FUNCTION_BLOCK FB_FMS205_F2SeqPrep_SFC EXTENDS FB_ControllerBase_SFC
// Girar 8 veces el plato para determinar qué tipo de tapa hay en cada sector del plato

VAR_IN_OUT
	Medid			: FB_MedidorTapa;
	Induc		 	: FB_CaptadorInductivo;
	Fotoe			: FB_DetectorFotoelectrico;
	Plato			: FB_PlatoDivisor;
END_VAR

VAR
	Giros 			: INT := 0;
END_VAR

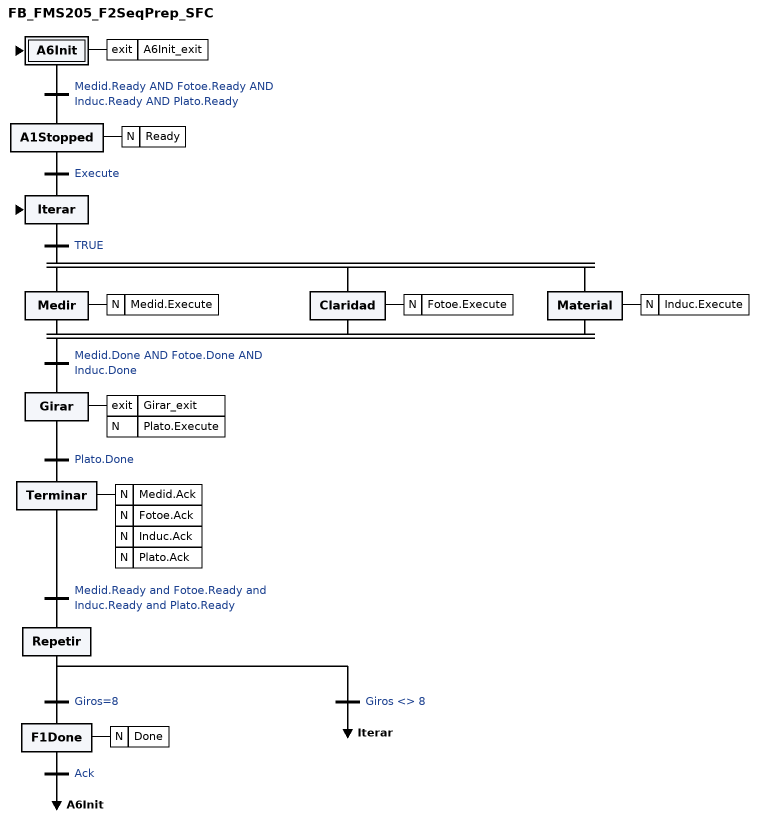
INITIAL_STEP A6Init:
    A6Init_exit(P0);  // exit action
END_STEP
TRANSITION FROM A6Init TO A1Stopped
    := Medid.Ready AND Fotoe.Ready AND Induc.Ready AND Plato.Ready;
END_TRANSITION
STEP A1Stopped:
    Ready(N);
END_STEP
TRANSITION FROM A1Stopped TO Iterar
    := Execute;
END_TRANSITION
STEP Iterar:
END_STEP
TRANSITION FROM Iterar TO (Medir, Claridad, Material)
    := TRUE;
END_TRANSITION
STEP Medir:
    Medid.Execute(N);
END_STEP
STEP Claridad:
    Fotoe.Execute(N);
END_STEP
STEP Material:
    Induc.Execute(N);
END_STEP
TRANSITION FROM (Medir, Claridad, Material) TO Girar
    := Medid.Done AND Fotoe.Done AND Induc.Done;
END_TRANSITION
STEP Girar:
    Girar_exit(P0);  // exit action
    Plato.Execute(N);
END_STEP
TRANSITION FROM Girar TO Terminar
    := Plato.Done;
END_TRANSITION
STEP Terminar:
    Medid.Ack(N);
    Fotoe.Ack(N);
    Induc.Ack(N);
    Plato.Ack(N);
END_STEP
TRANSITION FROM Terminar TO Repetir
    := Medid.Ready and Fotoe.Ready and Induc.Ready and Plato.Ready;
END_TRANSITION
STEP Repetir:
END_STEP
TRANSITION FROM Repetir TO F1Done
    := Giros=8;
END_TRANSITION
STEP F1Done:
    Done(N);
END_STEP
TRANSITION FROM F1Done TO A6Init
    := Ack;
END_TRANSITION
TRANSITION FROM Repetir TO Iterar
    := Giros <> 8;
END_TRANSITION

ACTION A6Init_exit:
Giros:=0;
END_ACTION

ACTION Girar_exit:
Giros:=Giros+1;
END_ACTION

END_FUNCTION_BLOCK

(* stored: Version 1.1.0.1, ProductVersion 3.1.4024.11
   POU FB_FMS205_F2SeqPrep_SFC: Id {306e8fb2-9473-4dd1-ac8a-7196779de084}, SpecialFunc None
   Action A6Init_exit: Id {e1190fd2-b61b-4572-abcd-f44d34d42ffc}
   Action Girar_exit: Id {50a4a834-adbe-40c6-b72d-eb4caaf0978f} *)
